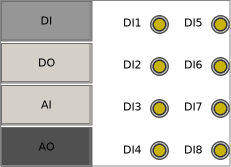
VISUALIZATION Digital_Inputs  // 231x167
    Button (1,127 91x40), "AO"
        OnMouseUp: change screen: Analog_Outputs
    Button (1,1 91x40), "DI"
        OnMouseUp: change screen: Digital_Inputs
    Button (1,43 91x40), "DO"
        OnMouseDown: change screen: Digital_Outputs
        OnMouseUp: change screen: Digital_Outputs
    Button (1,85 91x40), "AI"
        OnMouseUp: change screen: Analog_Inputs
    Lamp1 (149,14 21x21), variable: GVL_IO.DI1, style: Lamp-Lamp1-Yellow
    Lamp1 (149,56 21x21), variable: GVL_IO.DI2, style: Lamp-Lamp1-Yellow
    Lamp1 (149,98 21x21), variable: GVL_IO.DI3, style: Lamp-Lamp1-Yellow
    Lamp1 (149,140 21x21), variable: GVL_IO.DI4, style: Lamp-Lamp1-Yellow
    Label (113,8 39x30), "DI1"
    Label (113,50 39x30), "DI2"
    Label (113,92 39x30), "DI3"
    Label (113,135 39x30), "DI4"
    Lamp1 (210,14 21x21), variable: GVL_IO.DI5, style: Lamp-Lamp1-Yellow
    Lamp1 (210,56 21x21), variable: GVL_IO.DI6, style: Lamp-Lamp1-Yellow
    Lamp1 (210,98 21x21), variable: GVL_IO.DI7, style: Lamp-Lamp1-Yellow
    Lamp1 (210,140 21x21), variable: GVL_IO.DI8, style: Lamp-Lamp1-Yellow
    Label (174,8 39x30), "DI5"
    Label (174,50 39x30), "DI6"
    Label (174,92 39x30), "DI7"
    Label (174,135 39x30), "DI8"
END_VISUALIZATION

(* stored: Version 1.1.0.1, ProductVersion 3.1.4024.4
   Visu Digital_Inputs: Id {ca6391a7-78ec-4fed-aec4-081a50f0fd01} *)
